FUNCTION_BLOCK BLIND_SECURITY
  VAR_INPUT
    UP : BOOL;
    DN : BOOL;
    S_IN : BYTE;
    PI : BYTE;
    AI : BYTE;
    FIRE : BOOL;
    WIND : BOOL;
    ALARM : BOOL;
    DOOR : BOOL;
    RAIN : BOOL;
    {attribute 'input_constant'}
    Alarm_UP : BOOL := TRUE;
    {attribute 'input_constant'}
    WIND_UP : BOOL := TRUE;
    {attribute 'input_constant'}
    RAIN_UP : BOOL := FALSE;
  END_VAR
  VAR_OUTPUT
    QU : BOOL;
    QD : BOOL;
    STATUS : BYTE;
    PO : BYTE;
    AO : BYTE;
  END_VAR

            IF Fire THEN
	QU := TRUE;
	QD := FALSE;
	status := 111;
ELSIF Wind THEN
	QU := Wind_up;
	QD := NOT wind_up;
	status := 112;
ELSIF alarm THEN
	QU := Alarm_up;
	QD := NOT Alarm_up;
	status := 113;
ELSIF Door THEN
	QU := TRUE;
	QD := FALSE;
	status := 114;
ELSIF Rain AND NOT (up XOR dn) THEN
	QU := rain_up;
	QD := NOT rain_up;
	status := 115;
ELSE
	QU := UP;
	QD := DN;
	status := S_IN;
	po := pi;
	ao := ai;
END_IF;


(* revision history
hm	29. sep 2007	rev 1.0
	original release

hm	6. oct 2007		rev 1.1
	added pos and angle inputs and outputs
	manual will override rain position
	alarm position can now be configured

hm		12. feb. 2008	rev 1.2
	added config variables rain_up and wind_up
	position for rain and wind is now configurable
*)


          
END_FUNCTION_BLOCK

FUNCTION_BLOCK BLIND_SET
  VAR_INPUT
    UP : BOOL;
    DN : BOOL;
    S_IN : BYTE;
    PI : BYTE;
    AI : BYTE;
    IN : BOOL;
    PX : BYTE;
    AX : BYTE;
    {attribute 'input_constant'}
    OVERRIDE_MANUAL : BOOL;
    {attribute 'input_constant'}
    RESTORE_POSITION : BOOL;
    {attribute 'input_constant'}
    RESTORE_TIME : TIME := TIME#1m0s0ms;
  END_VAR
  VAR_OUTPUT
    QU : BOOL;
    QD : BOOL;
    STATUS : BYTE;
    PO : BYTE;
    AO : BYTE;
  END_VAR
  VAR
    tx : TIME;
    ps : BYTE;
    as : BYTE;
    last : TIME;
  END_VAR

            (* read system time *)
tx := DWORD_TO_TIME(OSCAT_BASIC.T_PLC_MS());

(* check inputs *)
IF IN THEN
	IF override_manual OR (UP AND DN) THEN
		status := 178;
	END_IF;
END_IF;

(* state machine *)
CASE STATUS OF
	0: (* power on state *)
		status := S_IN;

	178: (* force values from PX and AX *)
		PO := PX;
		AO := AX;
		QU := TRUE;
		QD := TRUE;
		(* check for end of forced position *)
		IF NOT in THEN
			STATUS := SEL(RESTORE_POSITION, S_IN, 179);
			last := tx;
		END_IF;

	179: (* restore previous position *)
		PO := ps;
		AO := as;
		IF ((PO = PI) AND (AO = AI))  OR tx - last >= RESTORE_TIME THEN
			status := S_IN;
		END_IF;

ELSE
	(* no operation transfer inputs to outputs *)
	PO := PI;
	ps := PI;
	AO := AI;
	as := AI;
	STATUS := S_IN;
	QU := UP;
	QD := DN;
END_CASE;


(* revision history
hm	27. jul 2009	rev 1.0
	original release

*)
          
END_FUNCTION_BLOCK

FUNCTION_BLOCK BLIND_SHADE
  VAR_INPUT
    UP : BOOL;
    DN : BOOL;
    S_IN : BYTE;
    PI : BYTE;
    AI : BYTE;
    ENABLE : BOOL;
    SUN : BOOL;
  END_VAR
  VAR_IN_OUT
    CX : OSCAT_BASIC.CALENDAR;
  END_VAR
  VAR_INPUT
    {attribute 'input_constant'}
    sunrise_offset : TIME := TIME#60m0s0ms;
    {attribute 'input_constant'}
    sunset_preset : TIME := TIME#60m0s0ms;
    {attribute 'input_constant'}
    direction : REAL := 180;
    {attribute 'input_constant'}
    angle_offset : REAL := 80;
    {attribute 'input_constant'}
    slat_width : REAL := 80;
    {attribute 'input_constant'}
    Slat_spacing : REAL := 60;
    {attribute 'input_constant'}
    Shade_delay : TIME := TIME#1m0s0ms;
    {attribute 'input_constant'}
    Shade_pos : BYTE;
  END_VAR
  VAR_OUTPUT
    QU : BOOL;
    QD : BOOL;
    STATUS : BYTE;
    PO : BYTE;
    AO : BYTE;
  END_VAR
  VAR
    angle : REAL;
    sun_delay : OSCAT_BASIC.TOF;
  END_VAR

            (* the input sun is sent through tof which will delay the shade for the time shade_delay *)
sun_delay(IN := sun, PT := shade_delay);

IF UP AND DN AND enable AND sun_delay.Q AND cx.SUN_HOR > direction - angle_offset AND cx.SUN_HOR < direction + angle_offset AND
	DT_TO_TOD(cx.UTC) > cx.SUN_RISE + sunrise_offset AND DT_TO_TOD(cx.UTC) < cx.SUN_SET - sunset_preset THEN
	status := 151;
	QU := UP;
	QD := DN;
	(* position is predefined *)
	po := shade_pos;
	(* shading is active now calculate the slat angle *)
	(* calculate the max angle for the blind *)
	angle := OSCAT_BASIC.DEG(ATAN(slat_spacing / slat_width));
	(* check if sun angle is between 0 and max angle *)
	IF cx.SUN_VER > 0.0 AND cx.SUN_VER < angle THEN
		angle := cx.SUN_VER + OSCAT_BASIC.DEG(ACOS(COS(OSCAT_BASIC.RAD(cx.SUN_VER))*slat_spacing / Slat_width));
		ao := INT_TO_BYTE(DINT_TO_INT(LIMIT(0,TRUNC(angle * 2.833333333), 255)));
	ELSE
		ao := 255;
	END_IF;
ELSE
	QU := UP;
	QD := DN;
	po := pi;
	ao := ai;
	status := S_IN;
END_IF;

(* revision history
hm	15 oct. 2007	rev 1.0
	original version

hm	19. oct 2007	rev 1.1
	manual mode was not detected because outputs were checked and not inputs UP and DN

hm	24. nov 2007	rev 1.2
	added shade_delay to avoid constant up and down if sun is out parcially

hm	8. feb 2009	rev 1.3
	added shading position shade_pos to be configured
	changed inputs to utilize calendar data structure

hm	13. mar. 2009	rev 1.4
	improved code

*)
          
END_FUNCTION_BLOCK

FUNCTION_BLOCK BLIND_SHADE_S
  VAR_INPUT
    UP : BOOL;
    DN : BOOL;
    S_IN : BYTE;
    PI : BYTE;
    ENABLE : BOOL;
    SUN : BOOL;
    HORZ1 : REAL := 100;
    HORZ2 : REAL := 260;
    VERT : REAL := 90;
    ALERT : BOOL := FALSE;
  END_VAR
  VAR_IN_OUT
    CX : OSCAT_BASIC.calendar;
  END_VAR
  VAR_INPUT
    {attribute 'input_constant'}
    sunrise_offset : TIME := TIME#60m0s0ms;
    {attribute 'input_constant'}
    sunset_preset : TIME := TIME#60m0s0ms;
    {attribute 'input_constant'}
    shade_delay : TIME := TIME#1m0s0ms;
    {attribute 'input_constant'}
    shade_pos : BYTE;
  END_VAR
  VAR_OUTPUT
    QU : BOOL;
    QD : BOOL;
    STATUS : BYTE;
    PO : BYTE;
  END_VAR
  VAR
    sun_delay : OSCAT_BASIC.TOF;
  END_VAR

            (* status definition
   151 = shadow               move shutter down for shadowing
   152 = alert                  move shutter up by setting QU:=TRUE when door is open.
*)

(* the input sun is sent through tof which will delay the shade for the time shade_delay *)
sun_delay(IN := sun, PT := shade_delay);

IF ALERT THEN
   QU := TRUE;
   QD := FALSE;
   STATUS := 152;
ELSIF UP AND DN AND ENABLE AND sun_delay.Q
AND (CX.SUN_HOR > HORZ1) AND (CX.SUN_HOR < HORZ2)
AND (CX.SUN_VER < VERT)
AND (DT_TO_TOD(CX.UTC) > CX.SUN_RISE + sunrise_offset) AND (DT_TO_TOD(CX.UTC) < CX.SUN_SET - sunset_preset) THEN
   QU := UP;
   QD := DN;
   STATUS := 151;
   (* Calculate Position, must be shade_pos or less *)
   PO := MIN(PI, shade_pos);
ELSE
   QU := UP;
   QD := DN;
   PO := PI;
   STATUS := S_IN;
END_IF;



(* revision history
hf	12 nov. 2009	rev 1.0
	original version

*)
          
END_FUNCTION_BLOCK

FUNCTION BUILDING_VERSION : DWORD
  VAR_INPUT
    IN : BOOL;
  END_VAR

            IF in THEN
	BUILDING_VERSION := DATE_TO_DWORD(D#2011-02-3);
ELSE
	BUILDING_VERSION := 100;
END_IF;

(* revision history
hm	6. oct 2006	rev 1.0
	original version

hm	16. dec 2007	rev 1.1
	added possibility to return date and version depending on IN.

*)
          
END_FUNCTION
